(* CODESYS project FU_lwBitPart.xml

Project tree, tasks and I/O mapping:
  function FU_lwBitPart [ST]
*)

// FU_lwBitPart
//This function changed only the needed bits of a variable
// |**Version**|**Author**| **Date** |**Changes**
// | 1         | NSN      | 16-03-22 | Creation
FUNCTION FU_lwBitPart : BOOL
VAR_IN_OUT
	valueChange		:LWORD;		//Variable to change
END_VAR
VAR_INPUT
	value			:LWORD;		//Value to change bits to
	amount			:BYTE;		//Amount of bits to change
	offset			:BYTE;		//Offset in variable to change bits at
END_VAR

valueChange		:=		(valueChange AND ROL(GConstants.binaryInvMaskLWord[amount],offset)) OR SHL(value AND GConstants.binaryMaskLWord[amount],offset);

END_FUNCTION
